PROGRAM MAIN
VAR
	Counter: INT;
END_VAR

Counter:=Counter+1;

END_PROGRAM

(* stored: Version 1.1.0.1, ProductVersion 3.1.4024.11
   POU MAIN: Id {a006fe57-da36-4aba-b269-66eb17a3ab15}, SpecialFunc None *)
